(* PLC project Unnamed, Unknown Unnamed 1 *)
(* stored: creationDateTime 2023-03-27T22:02:19, modificationDateTime 2023-05-17T20:40:07 *)

PROGRAM program0
  VAR_EXTERNAL
    start : BOOL;  (* press to start *)
    stop : BOOL;  (* stop all progress *)
  END_VAR
  VAR
    cncsen1 AT %IX100.2 : BOOL;  (* sensor for base production *)
    cncsen2 AT %IX100.3 : BOOL;  (* sensor for base production *)
    cncsen1B AT %IX100.4 : BOOL;  (* sensor for lid production *)
    cncsen2B AT %IX100.5 : BOOL;  (* sensor for lid production *)
    mchnsts AT %IX100.6 : BOOL;  (* gather machine status for raw material feed *)
    mchnsts2 AT %IX100.7 : BOOL;  (* gather machine status for raw material feed *)
    rdrctsns AT %IX101.0 : BOOL;  (* sensor pusher :D *)
    sensor1greenlid AT %IX101.4 : BOOL;  (* gather machine status for raw material feed *)
    sensor2greenbase AT %IX101.5 : BOOL;  (* gather machine status for raw material feed *)
    sensor1bluelid AT %IX101.6 : BOOL;  (* gather machine status for raw material feed *)
    sensor2bluebase AT %IX101.7 : BOOL;  (* gather machine status for raw material feed *)
    rstcnt AT %IX102.0 : BOOL;  (* gather machine status for raw material feed *)
    lids AT %QX100.0 : BOOL;  (* ask machine to produce lids *)
    cnccon1 AT %QX100.2 : BOOL;  (* conveyor control for machine feed *)
    cnccon2 AT %QX100.3 : BOOL;  (* conveyor control for machine feed *)
    cnc1 AT %QX100.7 : BOOL;  (* start machine *)
    cnc2 AT %QX101.0 : BOOL;  (* start machine *)
    rdrct AT %QX101.2 : BOOL;  (* pusher :D *)
    clampgreenlid AT %QX101.6 : BOOL;  (* pengaturan clamp green lid *)
    clampgreenbase AT %QX101.7 : BOOL;  (* pengaturan clamp green base *)
    clampgreenrise AT %QX102.0 : BOOL;  (* pengaturan clamp green base *)
    clamplidblue AT %QX102.1 : BOOL;  (* pengaturan clamp green base *)
    clampbaseblue AT %QX102.2 : BOOL;  (* pengaturan clamp green base *)
    clampbluerise AT %QX102.3 : BOOL;  (* pengaturan clamp green base *)
    picker1z AT %QX102.4 : BOOL;  (* pengaturan clamp green base *)
    picker1x AT %QX102.5 : BOOL;  (* pengaturan clamp green base *)
    picker1G AT %QX102.6 : BOOL;  (* pengaturan clamp green base *)
    picker2z AT %QX102.7 : BOOL;  (* pengaturan clamp green base *)
    picker2x AT %QX103.0 : BOOL;  (* pengaturan clamp green base *)
    picker2g AT %QX103.1 : BOOL;  (* pengaturan clamp green base *)
    conveyorpck AT %QX103.2 : BOOL;  (* pengaturan clamp green base *)
    VIR1 AT %QX0.0 : BOOL;  (* virtual output for machine base *)
    VIR2 AT %QX0.1 : BOOL;  (* virtual output for machine base *)
    VIR3 AT %QX0.2 : BOOL;  (* virtual output for machine lid *)
    VIR4 AT %QX0.3 : BOOL;  (* virtual output for machine lid *)
    VIR5 AT %QX0.4 : BOOL;  (* virtual output for machine lid *)
    VIR6 AT %QX0.5 : BOOL;  (* virtual output for machine lid *)
    VIR7 AT %QX0.6 : BOOL;  (* virtual output for machine lid *)
    VIR8 AT %QX0.7 : BOOL;  (* virtual output for machine lid *)
    VIR9 AT %QX1.0 : BOOL;  (* virtual output for machine lid *)
    VIR10 AT %QX1.1 : BOOL;  (* virtual output for machine lid *)
    VIR11 AT %QX1.2 : BOOL;  (* virtual output for machine lid *)
    VIR12 AT %QX1.3 : BOOL;  (* virtual output for machine lid *)
    VIR13 AT %QX2.4 : BOOL;  (* virtual output for machine lid *)
  END_VAR
  VAR
    cncton1 : TON;  (* counter for machine *)
    cncton2 : TON;  (* counter for machine lid *)
    cncton3 : TON;
    cncton4 : TON;
    cncton5 : TON;
    cncton6 : TON;
    cncton7 : TON;
    cncton8 : TON;
    cncton9 : TON;
    cncton10 : TON;
    cncton11 : TON;
    cncton12 : TON;
    cncton13 : TON;
    cncton14 : TON;
    CTU0 : CTU;
  END_VAR
  VAR  (* added by the conversion: wires and edge detectors of the diagram *)
    R_TRIG1 : R_TRIG;
  END_VAR

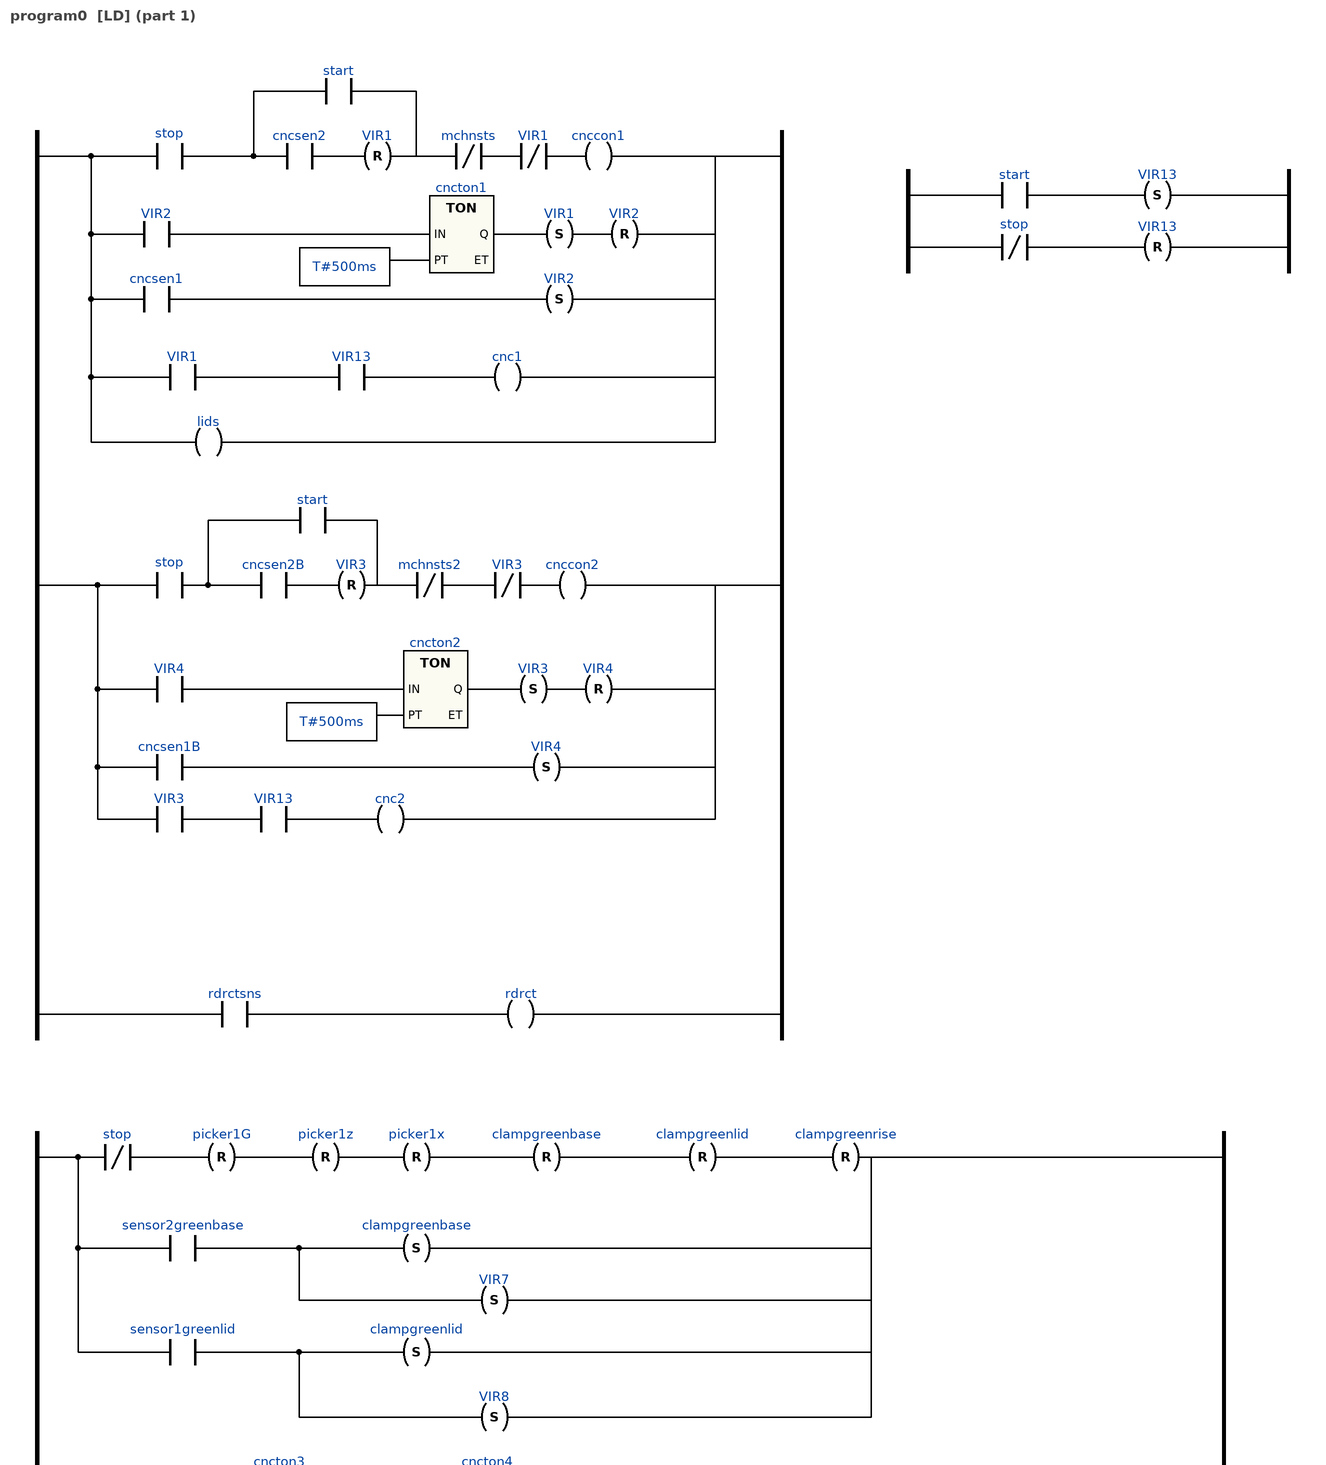
(* LD diagram, written out as Structured Text *)
IF stop AND cncsen2 THEN VIR1 := FALSE; END_IF;
cnccon1 := stop AND (cncsen2 OR start) AND NOT mchnsts AND NOT VIR1;
IF start THEN VIR13 := TRUE; END_IF;
cncton1(IN := VIR2, PT := T#500ms);
IF cncton1.Q THEN VIR1 := TRUE; END_IF;
IF cncton1.Q THEN VIR2 := FALSE; END_IF;
IF NOT stop THEN VIR13 := FALSE; END_IF;
IF cncsen1 THEN VIR2 := TRUE; END_IF;
cnc1 := VIR1 AND VIR13;
lids := TRUE;
IF stop AND cncsen2B THEN VIR3 := FALSE; END_IF;
cnccon2 := stop AND (cncsen2B OR start) AND NOT mchnsts2 AND NOT VIR3;
cncton2(IN := VIR4, PT := T#500ms);
IF cncton2.Q THEN VIR3 := TRUE; END_IF;
IF cncton2.Q THEN VIR4 := FALSE; END_IF;
IF cncsen1B THEN VIR4 := TRUE; END_IF;
cnc2 := VIR3 AND VIR13;
rdrct := rdrctsns;
IF NOT stop THEN picker1G := FALSE; END_IF;
IF NOT stop THEN picker1z := FALSE; END_IF;
IF NOT stop THEN picker1x := FALSE; END_IF;
IF NOT stop THEN clampgreenbase := FALSE; END_IF;
IF NOT stop THEN clampgreenlid := FALSE; END_IF;
IF NOT stop THEN clampgreenrise := FALSE; END_IF;
IF sensor2greenbase THEN clampgreenbase := TRUE; END_IF;
IF sensor2greenbase THEN VIR7 := TRUE; END_IF;
IF sensor1greenlid THEN clampgreenlid := TRUE; END_IF;
IF sensor1greenlid THEN VIR8 := TRUE; END_IF;
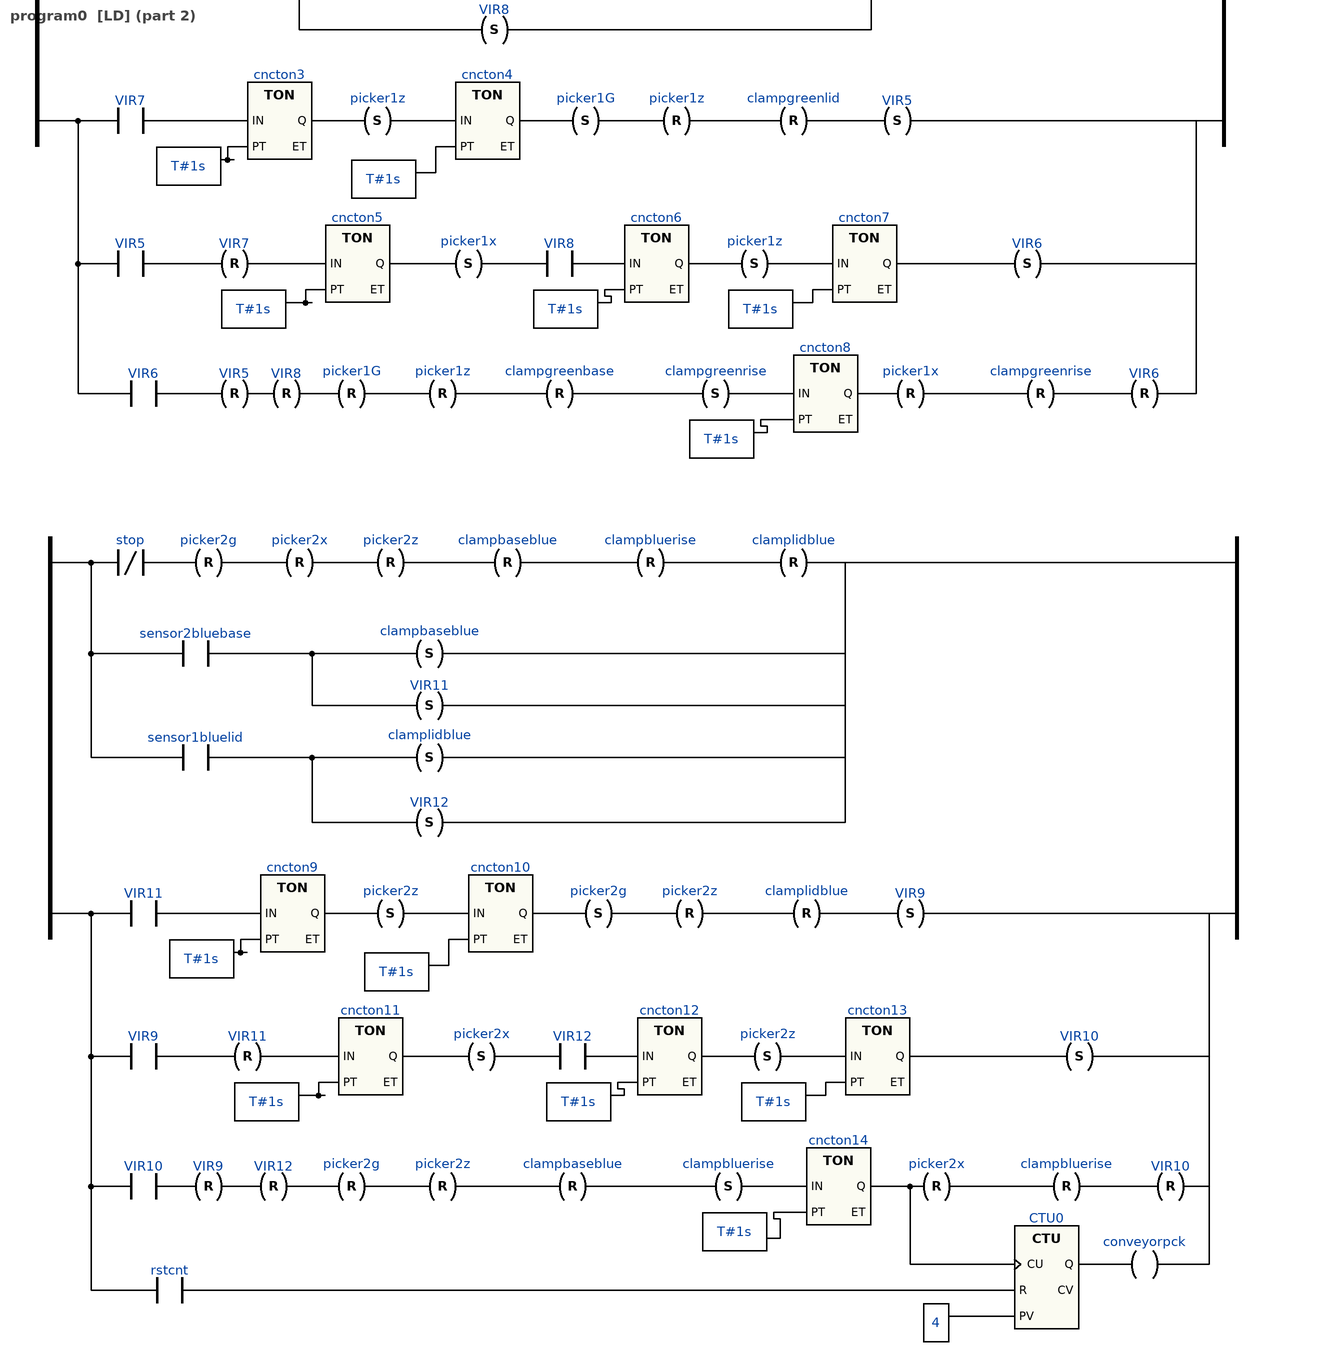
cncton3(IN := VIR7, PT := T#1s);
IF cncton3.Q THEN picker1z := TRUE; END_IF;
cncton4(IN := cncton3.Q, PT := T#1s);
IF cncton4.Q THEN picker1G := TRUE; END_IF;
IF cncton4.Q THEN picker1z := FALSE; END_IF;
IF cncton4.Q THEN clampgreenlid := FALSE; END_IF;
IF cncton4.Q THEN VIR5 := TRUE; END_IF;
IF VIR5 THEN VIR7 := FALSE; END_IF;
cncton5(IN := VIR5, PT := T#1s);
IF cncton5.Q THEN picker1x := TRUE; END_IF;
cncton6(IN := cncton5.Q AND VIR8, PT := T#1s);
IF cncton6.Q THEN picker1z := TRUE; END_IF;
cncton7(IN := cncton6.Q, PT := T#1s);
IF cncton7.Q THEN VIR6 := TRUE; END_IF;
IF VIR6 THEN VIR5 := FALSE; END_IF;
IF VIR6 THEN VIR8 := FALSE; END_IF;
IF VIR6 THEN picker1G := FALSE; END_IF;
IF VIR6 THEN picker1z := FALSE; END_IF;
IF VIR6 THEN clampgreenbase := FALSE; END_IF;
IF VIR6 THEN clampgreenrise := TRUE; END_IF;
cncton8(IN := VIR6, PT := T#1s);
IF cncton8.Q THEN picker1x := FALSE; END_IF;
IF cncton8.Q THEN clampgreenrise := FALSE; END_IF;
IF cncton8.Q THEN VIR6 := FALSE; END_IF;
IF NOT stop THEN picker2g := FALSE; END_IF;
IF NOT stop THEN picker2x := FALSE; END_IF;
IF NOT stop THEN picker2z := FALSE; END_IF;
IF NOT stop THEN clampbaseblue := FALSE; END_IF;
IF NOT stop THEN clampbluerise := FALSE; END_IF;
IF NOT stop THEN clamplidblue := FALSE; END_IF;
IF sensor2bluebase THEN clampbaseblue := TRUE; END_IF;
IF sensor2bluebase THEN VIR11 := TRUE; END_IF;
IF sensor1bluelid THEN clamplidblue := TRUE; END_IF;
IF sensor1bluelid THEN VIR12 := TRUE; END_IF;
cncton9(IN := VIR11, PT := T#1s);
IF cncton9.Q THEN picker2z := TRUE; END_IF;
cncton10(IN := cncton9.Q, PT := T#1s);
IF cncton10.Q THEN picker2g := TRUE; END_IF;
IF cncton10.Q THEN picker2z := FALSE; END_IF;
IF cncton10.Q THEN clamplidblue := FALSE; END_IF;
IF cncton10.Q THEN VIR9 := TRUE; END_IF;
IF VIR9 THEN VIR11 := FALSE; END_IF;
cncton11(IN := VIR9, PT := T#1s);
IF cncton11.Q THEN picker2x := TRUE; END_IF;
cncton12(IN := cncton11.Q AND VIR12, PT := T#1s);
IF cncton12.Q THEN picker2z := TRUE; END_IF;
cncton13(IN := cncton12.Q, PT := T#1s);
IF cncton13.Q THEN VIR10 := TRUE; END_IF;
IF VIR10 THEN VIR9 := FALSE; END_IF;
IF VIR10 THEN VIR12 := FALSE; END_IF;
IF VIR10 THEN picker2g := FALSE; END_IF;
IF VIR10 THEN picker2z := FALSE; END_IF;
IF VIR10 THEN clampbaseblue := FALSE; END_IF;
IF VIR10 THEN clampbluerise := TRUE; END_IF;
cncton14(IN := VIR10, PT := T#1s);
IF cncton14.Q THEN picker2x := FALSE; END_IF;
IF cncton14.Q THEN clampbluerise := FALSE; END_IF;
IF cncton14.Q THEN VIR10 := FALSE; END_IF;
R_TRIG1(CLK := cncton14.Q);
CTU0(CU := R_TRIG1.Q, R := rstcnt, PV := 4);
conveyorpck := CTU0.Q;
END_PROGRAM

PROGRAM warehouse
  VAR_EXTERNAL
    start : BOOL;
    stop : BOOL;
  END_VAR
  VAR
    Reset AT %IX102.1 : BOOL;
    Sensor AT %IX102.2 : BOOL;
    X AT %IX102.3 : BOOL;
    Z AT %IX102.4 : BOOL;
    sensorstrt AT %IX102.5 : BOOL;
    EntryCon AT %QX103.3 : BOOL;
    LoadCon AT %QX103.4 : BOOL;
    angkat AT %QX103.5 : BOOL;
    kiri AT %QX103.6 : BOOL;
    kanan AT %QX103.7 : BOOL;
    Target AT %QW100 : INT;
    DigitalDis AT %QW101 : INT;
    DigitalDis0 AT %QW102 : INT;
    VIR1 AT %QX1.4 : BOOL;
    VIR2 AT %QX1.5 : BOOL;
    VIR3 AT %QX1.6 : BOOL;
    VIR4 AT %QX1.7 : BOOL;
    VIR10 AT %QX2.1 : BOOL;
    VIRblokx AT %QX2.2 : BOOL;
    VIRblokz AT %QX2.3 : BOOL;
  END_VAR
  VAR
    TON0 : TON;
    TON1 : TON;
    CTU0 : CTU;
    TON2 : TON;
    TON7 : TON;
    TON4 : TON;
    TON6 : TON;
    TON3 : TON;
    CTU1 : CTU;
  END_VAR
  VAR  (* added by the conversion: wires and edge detectors of the diagram *)
    R_TRIG1 : R_TRIG;
    F_TRIG2 : F_TRIG;
    F_TRIG3 : F_TRIG;
    R_TRIG4 : R_TRIG;
    F_TRIG5 : F_TRIG;
    _AND69_OUT : BOOL;
  END_VAR

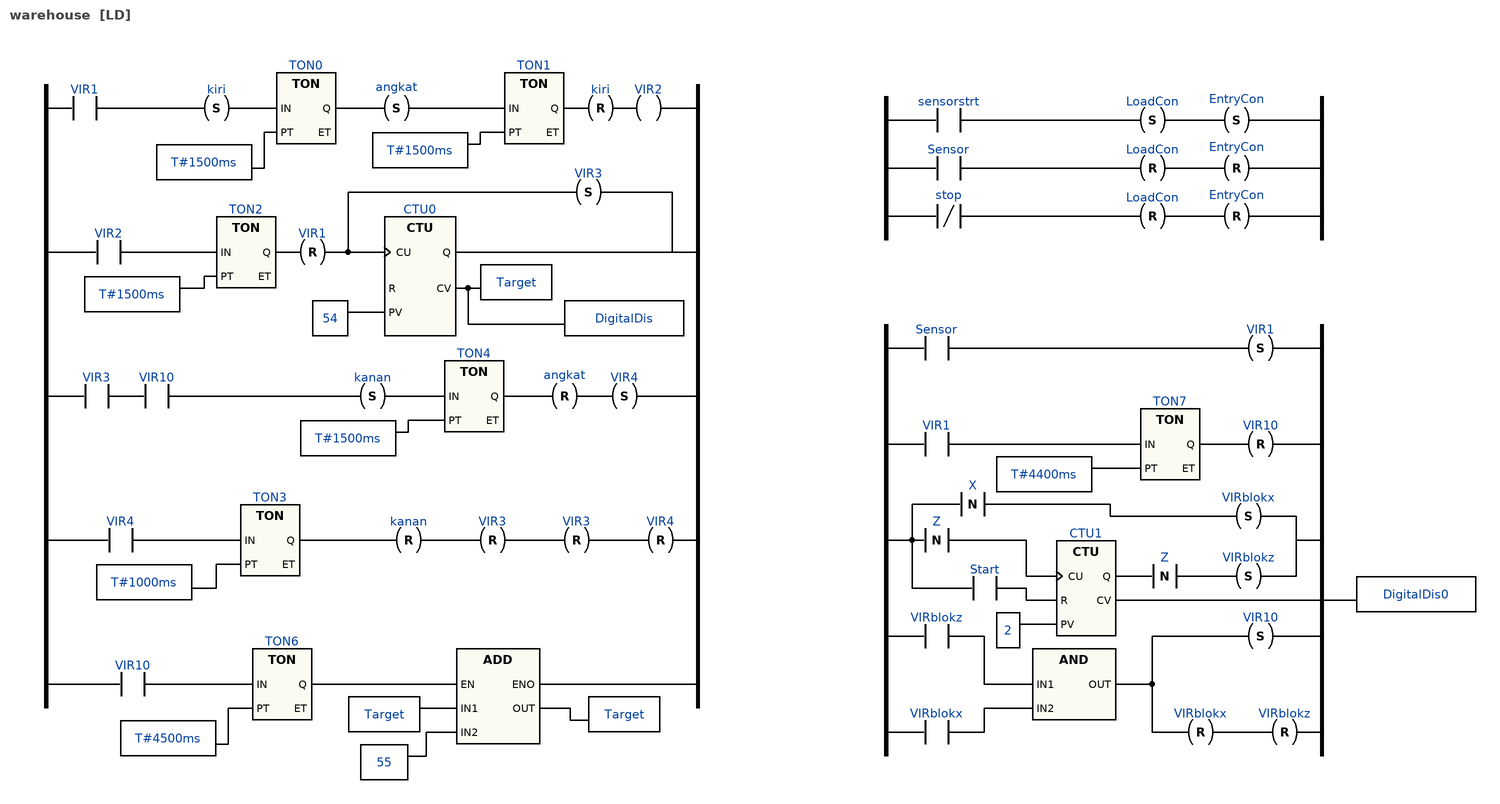
(* LD diagram, written out as Structured Text *)
IF VIR1 THEN kiri := TRUE; END_IF;
TON0(IN := VIR1, PT := T#1500ms);
IF TON0.Q THEN angkat := TRUE; END_IF;
TON1(IN := TON0.Q, PT := T#1500ms);
IF TON1.Q THEN kiri := FALSE; END_IF;
VIR2 := TON1.Q;
IF sensorstrt THEN LoadCon := TRUE; END_IF;
IF sensorstrt THEN EntryCon := TRUE; END_IF;
IF Sensor THEN LoadCon := FALSE; END_IF;
IF Sensor THEN EntryCon := FALSE; END_IF;
TON2(IN := VIR2, PT := T#1500ms);
IF TON2.Q THEN VIR3 := TRUE; END_IF;
IF NOT stop THEN LoadCon := FALSE; END_IF;
IF NOT stop THEN EntryCon := FALSE; END_IF;
IF TON2.Q THEN VIR1 := FALSE; END_IF;
R_TRIG1(CLK := TON2.Q);
CTU0(CU := R_TRIG1.Q, PV := 54);
Target := CTU0.CV;
DigitalDis := CTU0.CV;
IF Sensor THEN VIR1 := TRUE; END_IF;
IF VIR3 AND VIR10 THEN kanan := TRUE; END_IF;
TON4(IN := VIR3 AND VIR10, PT := T#1500ms);
IF TON4.Q THEN angkat := FALSE; END_IF;
IF TON4.Q THEN VIR4 := TRUE; END_IF;
TON7(IN := VIR1, PT := T#4400ms);
IF TON7.Q THEN VIR10 := FALSE; END_IF;
F_TRIG2(CLK := X);
IF F_TRIG2.Q THEN VIRblokx := TRUE; END_IF;
TON3(IN := VIR4, PT := T#1000ms);
IF TON3.Q THEN kanan := FALSE; END_IF;
IF TON3.Q THEN VIR3 := FALSE; END_IF;
IF TON3.Q THEN VIR3 := FALSE; END_IF;
IF TON3.Q THEN VIR4 := FALSE; END_IF;
F_TRIG3(CLK := Z);
R_TRIG4(CLK := F_TRIG3.Q);
CTU1(CU := R_TRIG4.Q, R := Start, PV := 2);
F_TRIG5(CLK := Z);
IF CTU1.Q AND F_TRIG5.Q THEN VIRblokz := TRUE; END_IF;
DigitalDis0 := CTU1.CV;
_AND69_OUT := VIRblokz AND VIRblokx;
IF _AND69_OUT THEN VIR10 := TRUE; END_IF;
TON6(IN := VIR10, PT := T#4500ms);
IF TON6.Q THEN Target := Target + 55; END_IF;
IF _AND69_OUT THEN VIRblokx := FALSE; END_IF;
IF _AND69_OUT THEN VIRblokz := FALSE; END_IF;
END_PROGRAM

PROGRAM conveyorz
  VAR_EXTERNAL
    start : BOOL;
    stop : BOOL;
  END_VAR
  VAR
    conveyor1 AT %QX104.0 : BOOL;
    conveyor2 AT %QX104.1 : BOOL;
    conveyor3 AT %QX104.2 : BOOL;
    conveyor4 AT %QX104.3 : BOOL;
    conveyor5 AT %QX104.4 : BOOL;
    conveyor6 AT %QX104.5 : BOOL;
    conveyor7 AT %QX104.6 : BOOL;
    conveyor8 AT %QX104.7 : BOOL;
    conveyor9 AT %QX105.0 : BOOL;
    conveyor10 AT %QX105.1 : BOOL;
    conveyor11 AT %QX105.2 : BOOL;
    conveyor12 AT %QX105.3 : BOOL;
    conveyor13 AT %QX105.4 : BOOL;
    VIR1 AT %QX2.5 : BOOL;
  END_VAR

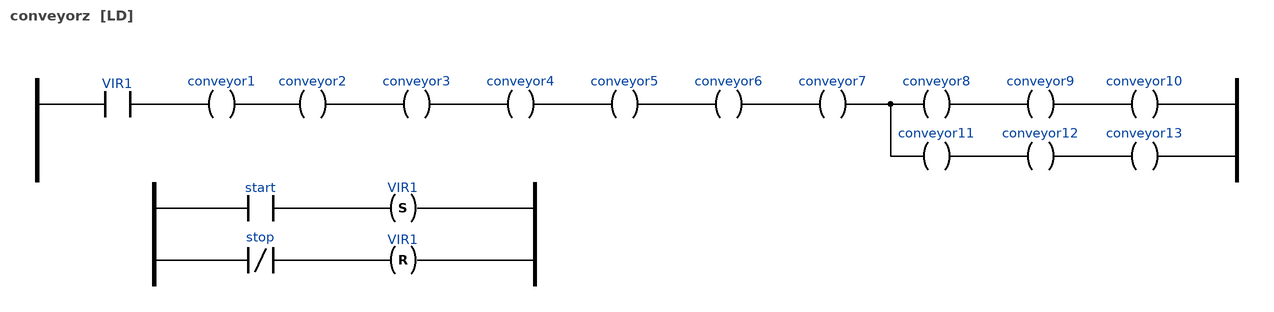
(* LD diagram, written out as Structured Text *)
conveyor1 := VIR1;
conveyor2 := VIR1;
conveyor3 := VIR1;
conveyor4 := VIR1;
conveyor5 := VIR1;
conveyor6 := VIR1;
conveyor7 := VIR1;
conveyor8 := VIR1;
conveyor9 := VIR1;
conveyor10 := VIR1;
conveyor11 := VIR1;
conveyor12 := VIR1;
conveyor13 := VIR1;
IF start THEN VIR1 := TRUE; END_IF;
IF NOT stop THEN VIR1 := FALSE; END_IF;
END_PROGRAM

CONFIGURATION Config0
  RESOURCE Res0 ON PLC
    VAR_GLOBAL
      start AT %IX100.0 : BOOL;
      stop AT %IX100.1 : BOOL;
    END_VAR
    TASK task0(INTERVAL := T#20ms, PRIORITY := 0);
    TASK task1(INTERVAL := T#20ms, PRIORITY := 0);
    TASK task2(INTERVAL := T#20ms, PRIORITY := 0);
    PROGRAM instance0 WITH task0 : program0;
    PROGRAM instance1 WITH task1 : warehouse;
    PROGRAM instance2 WITH task2 : conveyorz;
  END_RESOURCE
END_CONFIGURATION
